{attribute addProperty BoxType "EJ6002-0000-0016"}
{attribute addProperty Id "Transmit_requestBIT10.1251Receive_acceptedBIT10.1252Init_requestBIT10.1253Send_continuousBIT10.1254Output_lengthUSINT819"}
{attribute addProperty CRC "2534925159"}
{attribute addProperty SizeInBites "16"}
{attribute addProperty SizeInBytes "2"}
TYPE Ctrl_9717E367 :
STRUCT
	{attribute addProperty Name "Transmit_request"}
	Transmit_request : BIT;
	{attribute addProperty Name "Receive_accepted"}
	Receive_accepted : BIT;
	{attribute addProperty Name "Init_request"}
	Init_request : BIT;
	{attribute addProperty Name "Send_continuous"}
	Send_continuous : BIT;
	{attribute 'hide'}
	reserve_1_BIT_0 : BIT;
	{attribute 'hide'}
	reserve_1_BIT_1 : BIT;
	{attribute 'hide'}
	reserve_1_BIT_2 : BIT;
	{attribute 'hide'}
	reserve_1_BIT_3 : BIT;
	{attribute addProperty Name "Output_length"}
	Output_length : USINT;
END_STRUCT
END_TYPE

(* stored: Version 1.2.0.0, ProductVersion 3.1.4024.9
   DUT Ctrl_9717E367: Id {7b59baa0-d057-44a3-b839-6df5094acf0a} *)
